FUNCTION Convert_ULINT_TO_SINT : BOOL
VAR_INPUT
	in : ULINT;
	out : REFERENCE TO SINT;
END_VAR
VAR
	converted : SINT;
END_VAR

converted := ULINT_TO_SINT(in);

IF (SINT_TO_ULINT(converted) <> in) THEN
	RETURN;
END_IF

out := converted;
Convert_ULINT_TO_SINT := TRUE;

END_FUNCTION

(* stored: Version 1.1.0.1, ProductVersion 3.1.4024.12
   POU Convert_ULINT_TO_SINT: Id {91a96c45-ceef-446f-b0eb-22ff70e058b8}, SpecialFunc None *)
